{attribute 'qualified_only'}
{attribute 'strict'}
TYPE eState_Vertical :
(
	init := 0,
    checkPosition := 1,
    setPosition := 2,
    enableSpg := 3,
    confirmEnableSpg := 4,
    disableSpg := 5,
    confirmDisableSpg :=6,
    operation :=7
    
);
END_TYPE

(* stored: Version 1.1.0.1, ProductVersion 3.1.4024.11
   DUT eState_Vertical: Id {1fdeffad-8678-440d-bae5-75dbad51c410} *)
